// One event per notification, whatever the outcome - failures, errors, suite
// results and framework errors all raise exactly one.
//
// The IDs and severities differ per outcome so a filtered view can show suite
// results without every individual failure; what this checks is that each path
// reaches the logger and none raises twice.
FUNCTION_BLOCK TEST_EventReporterRaisesEachOutcomeOnce IMPLEMENTS I_Test
VAR
	Sink  : TestEventReporter;
	Tally : TestRunTally;
	ExpectedCount : UDINT;
	ActualCount	  : UDINT;
END_VAR

METHOD Run : BOOL
VAR_INPUT
	Enable : BOOL;
	Test   : I_TestAssertions;
END_VAR
Sink.TestFinished(SuiteLabel := 's', TestLabel := 'failed', Location := '',
				  Status := E_TestStatus.Failed, Kind := E_FailureKind.ValueMismatch,
				  Summary := 'x', ElapsedTime := 0.0, ElapsedCycles := 1, Assertions := 1);

Sink.TestFinished(SuiteLabel := 's', TestLabel := 'errored', Location := '',
				  Status := E_TestStatus.Errored, Kind := E_FailureKind.Environment,
				  Summary := 'y', ElapsedTime := 0.0, ElapsedCycles := 1, Assertions := 1);

Sink.FrameworkError(Source := 's', Message := 'something the framework could not do');

Tally.SetLabel('s');
Tally.Begin(2);
Tally.Record(Verdict := E_TestStatus.Passed, ElapsedTime := 0.1);
Tally.Record(Verdict := E_TestStatus.Failed, ElapsedTime := 0.1);
Tally.Finish();
Sink.SuiteFinished(Tally);
Sink.RunFinished(Status := Tally, TargetInfo := 'the verifier');

ExpectedCount := 5;
ActualCount	  := Sink.EventsSent;
Test.AssertEqual(ExpectedCount, ActualCount, 'five notifications, five events');

ExpectedCount := 0;
ActualCount	  := Sink.FailedSends;
Test.AssertEqual(ExpectedCount, ActualCount, 'none refused');

// A null status is refused rather than dereferenced, and raises nothing.
Sink.SuiteFinished(0);
Sink.RunFinished(Status := 0, TargetInfo := '');
ExpectedCount := 5;
ActualCount	  := Sink.EventsSent;
Test.AssertEqual(ExpectedCount, ActualCount, 'a null status raises nothing');

Run := TRUE;
END_METHOD

END_FUNCTION_BLOCK

(* stored: Version 1.1.0.1, ProductVersion 3.1.4026.18
   POU TEST_EventReporterRaisesEachOutcomeOnce: Id {9a3b3372-4b0e-445b-b143-6f9679d0c757}, SpecialFunc None
   Folder I_Test: Id {40670a9d-0990-492c-b427-87ba8a1140bd}
   Method Run: Id {4a043896-acc2-4f13-8cc1-b0b440b25e42} *)
